Fanuc KAREL source: KD00053.KL

PROGRAM KD00053
%NOLOCKGROUP
VAR
  I: INTEGER
  J: INTEGER
  B: BOOLEAN
  R: REAL
  S: STRING[80]
BEGIN
  I = J + 1
END KD00053
